FUNCTION_BLOCK fbUnderPresureTester_V2 IMPLEMENTS I_StationMachine
VAR_IN_OUT
	stInOuts 					: stUnderPressureTesterInOuts_V2;	//In Outs for modules
	stParams					: stUnderPressureTestParams_V2;		//Parameters for underpressure chamber
	stStatus					: stUnderPressureTestStatus_V2;		//Status struct
END_VAR
VAR_INPUT
END_VAR
VAR_OUTPUT
END_VAR
VAR
	fbVacuumMeasure				: 	fbAnalogMeasurement;		//Block for underpressure calibration
	fbTON_1Hz					: 	TON;						//Timer with 1 Hz cycle
	bOneHzClock					: 	BOOL;						//Bool variable for 1 Hz status
	iWorkStep					: 	INT;						//Step in sequence of work
	fbTON_VacumObtained			: 	TON;						//Filtering the vacuum status
	fbTON_VacumNearZero			: 	TON;						//Filtering the vacuum status
	I_PimSystem					: 	I_PIM;						//PIM block
	fbTON_VacuumMonitor			: 	TON;						//Checking that undeerpressure in increasing;			
	rLastUnderPressure			: 	REAL;						//Underpressure history		
	fbTOFF_CycleEndTurnOf		: 	TOF;						//Setting up end cycle
	//iCyclesToRepeat				: 	INT;						//How many cycles need to be done?		
	bServiceReset				: BOOL;							//Reset 
	bManual						: BOOL;							//Manual mode
END_VAR

ACT_Background();
CASE iWorkStep OF
	0:		// Init
		iWorkStep := 1;
		stInOuts.bPumpRly := FALSE;
		stInOuts.bEValve := TRUE;
		I_PimSystem.mSetNewMachineState(nPIM_MachineStates._0_Initialization);
	1:		// Wait for obtaining atmospheric pressure
		IF NOT stInOuts.bEValve THEN
			iWorkStep := 5;
		END_IF
	
	5:		// Setup new test
		I_PimSystem.mSetNewMachineState(nPIM_MachineStates._0_Standby_NotReady);
		iWorkStep := 10;
	10:		// Waiting for ext test premission 
		I_PimSystem.mSetNewMachineState(nPIM_MachineStates._2_ReadyForNewOperation);
		IF stInOuts.bLockSens AND stInOuts.bSafetyOK AND NOT stInOuts.bEValve AND stStatus.bWorkAllow THEN
			IF I_PimSystem.mSetNewMachineState(nPIM_MachineStates._3_NewOperationStarted) THEN
				iWorkStep := 15;
			END_IF
		END_IF
	15:		// Stating new cycle
		stInOuts.bPumpRly := TRUE;
		I_PimSystem.mSetNewMachineState(nPIM_MachineStates._4_OperationInProgress);
		iWorkStep := 20;
	20:		// Waiting for end of cycle
		IF fbTON_VacumObtained.Q THEN
			stInOuts.bPumpRly := FALSE;
			stInOuts.bEValve := TRUE;
			iWorkStep := 25;
		END_IF
	25:		//Waiting for pressure low value
		IF NOT stInOuts.bEValve THEN
			iWorkStep := 30;
		END_IF
	30:		//Waiting for doors open
		IF NOT stInOuts.bLockSens THEN
			iWorkStep := 5;
		END_IF
	50:		//Manual mode
		IF NOT stStatus.bManual THEN
			iWorkStep := 5;
		END_IF
	90:	//Error obtained
		I_PimSystem.mSetNewMachineState(nPIM_MachineStates._8_WaitForReset);
		iWorkStep	:= 91;
		stInOuts.bEValve	:= TRUE;
		stInOuts.bPumpRly	:= FALSE;
	91:	//Waiting for reset
		IF I_PimSystem.mSetNewMachineState(nPIM_MachineStates._9_ResetInProgress) OR bServiceReset THEN
			IF stInOuts.bSafetyOK THEN
				stInOuts.bEValve	:= TRUE;
				stInOuts.bPumpRly	:= FALSE;
				iWorkStep			:= 95;
			ELSE
				iWorkStep	:= 90;
			END_IF
		END_IF
	95:	//Reset confirmed
		I_PimSystem.mSetNewMachineState(nPIM_MachineStates._0_Standby_NotReady);
		iWorkStep		:= 5;
END_CASE

ACTION ACT_Background:
//------------------------------------------------------------------------------------------------
//Measurement scalling
fbVacuumMeasure(rIn:=stInOuts.iVacuumLevel,
				stMeasureScalingData:=stParams.stVacuumData,
				tStalaczasowa:= T#10MS,
				rOutFiltered=>stInOuts.rVacuumLevel);
//------------------------------------------------------------------------------------------------
//1Hz clock
fbTON_1Hz(IN:=NOT fbTON_1Hz.Q,PT:=T#500MS);
bOneHzClock := fbTON_1Hz.Q XOR bOneHzClock;
//------------------------------------------------------------------------------------------------
//LED Light Control
stInOuts.bLEDGreen		:= stStatus.bWorkEnd;
stInOuts.bLEDRed 		:= (NOT stInOuts.bSafetyOK AND bOneHzClock) OR stStatus.bError;
stInOuts.bLEDYellow 	:= (iWorkStep = 10) OR (stStatus.bBusy AND bOneHzClock) ;
stInOuts.bLEDReset 		:= NOT stInOuts.bSafetyOK;
//------------------------------------------------------------------------------------------------
//Vacuum obtained
fbTON_VacumObtained(IN:=stInOuts.rVacuumLevel>=stParams.rVaccumLevelToObtain,PT:=T#50MS);
//------------------------------------------------------------------------------------------------
//No Vacuum - Stable - Turn off 
fbTON_VacumNearZero(IN:=(stInOuts.rVacuumLevel<4), PT:= T#500MS);
stInOuts.bEValve R= fbTON_VacumNearZero.Q;
//------------------------------------------------------------------------------------------------
//Busy signal
stStatus.bBusy := stInOuts.bPumpRly;
//------------------------------------------------------------------------------------------------
//Checking increase of underpressure - Error
fbTON_VacuumMonitor(IN:=stStatus.bBusy AND (stInOuts.rVacuumLevel > rLastUnderPressure), PT:=T#5S);
//------------------------------------------------------------------------------------------------
//Calculating underpressure increasing
IF stInOuts.rVacuumLevel > rLastUnderPressure AND stStatus.bBusy THEN
	rLastUnderPressure := stInOuts.rVacuumLevel;
ELSIF NOT stStatus.bBusy THEN
	rLastUnderPressure := 0;
END_IF
//------------------------------------------------------------------------------------------------
// Cycle end status
fbTOFF_CycleEndTurnOf(IN:=fbTON_VacumObtained.Q,PT:=T#1S);
stStatus.bWorkEnd := fbTOFF_CycleEndTurnOf.Q;
//------------------------------------------------------------------------------------------------
// Error status setup
stStatus.bError := iWorkStep >= 90;
//------------------------------------------------------------------------------------------------
// Error pressure is no increasing 
IF fbTON_VacuumMonitor.Q AND NOT stStatus.bError THEN
	mNewEvent(nEventClass:=nPIM_EventClasses.Error,nEvent:=nUnderPressureTestErrorCodes.TestTimeOut);
END_IF
//------------------------------------------------------------------------------------------------
//Error safety turned on
IF NOT  stInOuts.bSafetyOK AND NOT stStatus.bError THEN
	mNewEvent(nEventClass:=nPIM_EventClasses.Error,nEvent:=nUnderPressureTestErrorCodes.SafetyError);
END_IF
//------------------------------------------------------------------------------------------------
END_ACTION

METHOD FB_init : BOOL
VAR_INPUT
	bInitRetains	: BOOL;
	bInCopyCode 	: BOOL;
	I_Pim			: I_PIM;
END_VAR
I_PimSystem := I_Pim;
END_METHOD

{warning 'add method implementation '}
(* Metoda TRUE kiedy dane wyjściowe są ok, jeśli nie FALSE (jeśli not bBusy i FALSE to błąd odczytu) *)
METHOD mGetParamsData : BOOL
VAR_INPUT
	(* Jeśli TRUE metoda okresla czy ma dostęp do parametrów, jeśli tak zwraca TRUE, jeśli nie FALSE*)
	bTestParams	: BOOL;
END_VAR
VAR_OUTPUT
	(* Maszyna odświeża dane*)
	bBusy	: BOOL;
	(* Wskaźnik do parametrów pracy maszyny*)
	pMachineParametersStruct	: POINTER TO BYTE;
	(* Rozmiar struktury parametrów pracy maszyny [bajty]*)
	uiMachineParametersSize	: UINT;
	(* Aktualna suma CRC16 obliczona z parametrów*)
	wActualCRC16SumInMachine	: WORD;
END_VAR
IF bTestParams THEN
	//mGetParamsData := stMachineSettings.bSerialCommunicationEN;
ELSE
	//pMachineParametersStruct := ADR(stParamAktProgramu);
	//uiMachineParametersSize := SIZEOF(stParamAktProgramu);
	wActualCRC16SumInMachine := F_DATA_TO_CRC16_CCITT(pData := pMachineParametersStruct, cbData := uiMachineParametersSize, crc := 16#0000);
	bBusy := FALSE;
	mGetParamsData := TRUE;	
END_IF
END_METHOD

METHOD INTERNAL mNewEvent : BOOL
VAR_INPUT
	nEventClass:nPIM_EventClasses;
	nEvent: nUnderPressureTestErrorCodes;
END_VAR
IF nEventClass = nPIM_EventClasses.AlarmAutoConfirm OR nEventClass = nPIM_EventClasses.Message THEN		// Alarm nieblokadowy
	I_PimSystem.mSetNewMachineState(nPIM_MachineStates._0_Initialization);
	iWorkStep := 90;
ELSE
	I_PimSystem.mSetNewMachineState(nPIM_MachineStates._7_ErrorOccurr);

	I_PimSystem.mNewEvent(iEventId := nEvent, nEventType := nEventClass, tMessageTime := T#0S);
	iWorkStep := 90;
END_IF
END_METHOD

END_FUNCTION_BLOCK

(* stored: Version 1.1.0.1, ProductVersion 3.1.4024.13
   POU fbUnderPresureTester_V2: Id {462e440b-7307-420e-9b04-0dfafe6159c5}, SpecialFunc None
   Action ACT_Background: Id {13628eb4-55a8-4aaa-a5cf-98a57b0ecf09}
   Method FB_init: Id {667e6daf-02d1-45ba-9492-c5dd84fa9c0d}
   Method mGetParamsData: Id {b52daad4-ffe4-4514-a088-af794b089f9c}
   Method mNewEvent: Id {1b4a9d77-38a3-427c-b260-2da22bfe9ca8} *)
